Fanuc KAREL source: ko00048.KL

-- PROVISIONAL review KL for V770-1; original PC SHA256 eb5de7ab0ac11a76ff6a460d948f2443385ef4cfbc95e6cffd507e3095913907
-- Incomplete behavior may be omitted. Consult companion uncertainty JSON. Do not deploy.
PROGRAM KO00048
%NOLOCKGROUP
BEGIN
  -- UNRESOLVED_PC offsets 5-12; opcodes 9D,23
  -- UNRESOLVED_PC offsets 17-69; opcodes 27,27,49,7E,AD,27,49,7E,AD,22,31,7E,4A
  -- UNRESOLVED_PC offsets 74-78; opcodes 7F
END KO00048
